FUNCTION_BLOCK "G152M_Code"
TITLE =G152M EXHAUST AIR LOUVER GERM 3
//COPYRIGHT:    (C) 2009  BUHLER AG, CH-9240 UZWIL, SWITZERLAND
//
//PRODUCT:      WinCoS_BIW01_09
//
//TITLE:        EXHAUST AIR LOUVER GERM 3
//                Machine group control
//                Maschinengruppensteuerung
//
//--------------------------------------------------------------------------------
//
//IDENT:        AUTHOR:             DEPT:                              DATE:
//
//P01_FB252.1.0 K.Renz              CSB41                              13.Jan.2010
//             1st Release
//
//--------------------------------------------------------------------------------
//
//PURPOSE:
//
//MANUAL :
//
//RESTRICTIONS:
//
//--------------------------------------------------------------------------------
AUTHOR : KR
FAMILY : USW
VERSION : 9.9


VAR
  Gr : "GCS7_GrpCtrlSub";	//Standard interface to group
  InOutValue1 : DINT ;	//Data for user
  InOutValue2 : DINT ;	//Data for user
  OutWayConflict : BOOL ;	//Data for user
  OutSelectionOk : BOOL ;	//Data for user
  CmdNewValue : BOOL ;	//Data for user
  CmdNewJob : BOOL ;	//Data for user
  OutCodeOK : BOOL ;	//Data for user
  InEndOfJob : BOOL ;	//Data for user
  staWayOk : BOOL ;	//Data for user
  EdgeStartRelease : BOOL ;	//Data for user
  USW8 : BOOL ;	//Data for user
  USW9 : BOOL ;	//Data for user
  USW10 : BOOL ;	//Data for user
  USW11 : BOOL ;	//Data for user
  USW12 : BOOL ;	//Data for user
  USW13 : BOOL ;	//Data for user
  USW14 : BOOL ;	//Data for user
  USW15 : BOOL ;	//Data for user
  A_2350_BZS01 : "GCS7_E_DigInput";	// DigInpCont
  A_2350_BZS02 : "GCS7_E_DigInput";	// DigInpCont
  A_2350_MXZ01 : "GCS7_E_ValveControl4Pos";	// VLS4Ctrl
END_VAR
VAR_TEMP
  tmpEnable : BOOL ;
  tmpFlag : BOOL ;
  tmpCmdNext : BOOL ;
  tmpLocal : BOOL ;
  tmpAspOk : BOOL ;
  tmpHWStop : BOOL ;
  tmpInstanzDBNo : INT ;
END_VAR
BEGIN
NETWORK
TITLE =



NETWORK
TITLE =Read command from group control
//Parameter
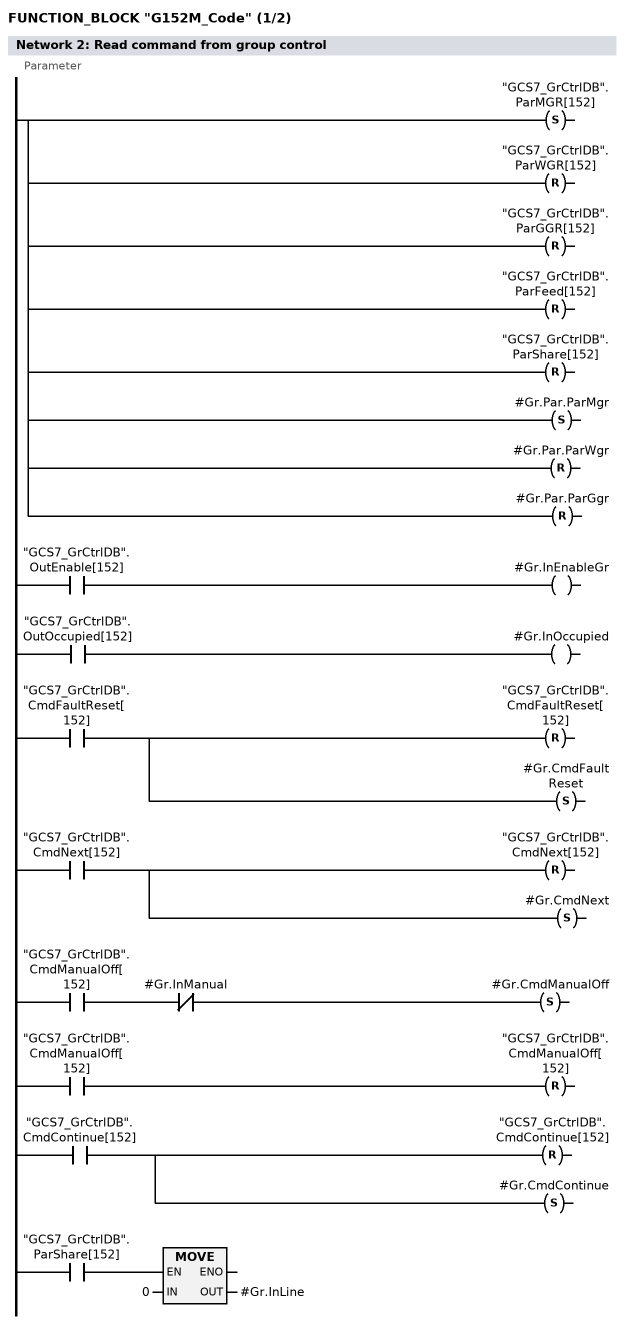
      SET   ;
      S     "GCS7_GrCtrlDB".ParMGR[152];
      R     "GCS7_GrCtrlDB".ParWGR[152];
      R     "GCS7_GrCtrlDB".ParGGR[152];
      R     "GCS7_GrCtrlDB".ParFeed[152];
      R     "GCS7_GrCtrlDB".ParShare[152];
      S     #Gr.Par.ParMgr;
      R     #Gr.Par.ParWgr;
      R     #Gr.Par.ParGgr;
//Command
      U     "GCS7_GrCtrlDB".OutEnable[152];
      =     #Gr.InEnableGr;
      U     "GCS7_GrCtrlDB".OutOccupied[152];
      =     #Gr.InOccupied;
      U     "GCS7_GrCtrlDB".CmdFaultReset[152];
      R     "GCS7_GrCtrlDB".CmdFaultReset[152];
      S     #Gr.CmdFaultReset;
      U     "GCS7_GrCtrlDB".CmdNext[152];
      R     "GCS7_GrCtrlDB".CmdNext[152];
      S     #Gr.CmdNext;

      U     "GCS7_GrCtrlDB".CmdManualOff[152];
      UN    #Gr.InManual;
      S     #Gr.CmdManualOff;
      U     "GCS7_GrCtrlDB".CmdManualOff[152];
      R     "GCS7_GrCtrlDB".CmdManualOff[152];

//      U     "GCS7_GrCtrlDB".CmdManualOff[152]
//      O     "GCS7_GrCtrlDB".OutOccupied[152]
//      R     "GCS7_GrCtrlDB".CmdManualOff[152]
//      S     #Gr.CmdManualOff

      U     "GCS7_GrCtrlDB".CmdContinue[152];
      R     "GCS7_GrCtrlDB".CmdContinue[152];
      S     #Gr.CmdContinue;
//Init Line Number
      U     "GCS7_GrCtrlDB".ParShare[152];
      SPBN  WE00;
      L     0;
      T     #Gr.InLine;
WE00: NOP   0;
NETWORK
TITLE =Call Methode Control
// 1. Handle Interface PCControl
// 2. Prepare mode --> ModePassive,ModeActive,ModeIdling
// 3. Reset global flags of the group
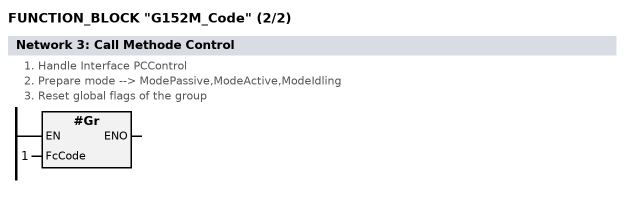
      CALL #Gr (
           FcCode                   := 1);
NETWORK
TITLE =Restart Idling Time

      L     #Gr.Par.ParIdling;
      L     2;
      >=I   ;
      SPB   IdTm;
      T     #Gr.Par.ParIdling;
IdTm: NOP   0;
      CLR   ;
      S     #Gr.CmdRestartIdling;
NETWORK
TITLE =Prepare global flags



NETWORK
TITLE =Set Pattern (Target position)

      U     #Gr.InManual;
      SPB   ILO6;
      L     0; // 0.0%
      O     "MAL1S019".PCRead.Step.StIdling;
      O     "MAL1S019".PCRead.Step.StPassive;
      SPB   PE;
      U     "MAL1S019Par".Par.FlagProcess.ProcessActive;
      O(    ;
      U     "MAL1S019Par".Par.FlagProcess.ProcessEnd; // germinating Process finished
      UN    "MAL1S019".PCRead.Step.StEmptying;
      )     ;
      SPBN  M003;
      NOP   0;
//BRT100310 - Abluftklappen haben gleichen Sollwert wie Frischluftklappen!
//      L     100                         // 100%
//      L     "MAL1S019Par".StepAct.PosWasteAirFlapBasic
//      -I
      L     "MAL1S019Par".Par.ParIntMachine.TargetPosFreshAir; //BRT100310
      L     "MAL1S019Par".Par.ParIntProcess.Value29; // Target Position FreshAir 2
      +I    ;
      L     2;
      /I    ;
      L     10; // convert to 0.1%
      *I    ;
PE:   NOP   0;

      U     "G152M".A_2350_MXZ01.InManual;
      SPB   Man1;
      T     #A_2350_MXZ01.InPositionMiddle; // setpoint element
Man1: NOP   0;

M003: NOP   0;
      SPA   En06;
ILO6: NOP   0;
//BRT100310      L     100                         // 100%
      L     "MAL1S019Par".Par.ParIntProcess.TarPos_ILO_FreshAir;
//BRT100310      -I
      L     10; // convert to 0.1%
      *I    ;
      T     #A_2350_MXZ01.InPositionMiddle; // setpoint element
En06: NOP   0;



NETWORK
TITLE =Interlocking WayOk



NETWORK
TITLE =Interlocking Autostart

      CLR   ;
      R     #Gr.OutAutostart;
NETWORK
TITLE =Interlocking Enable
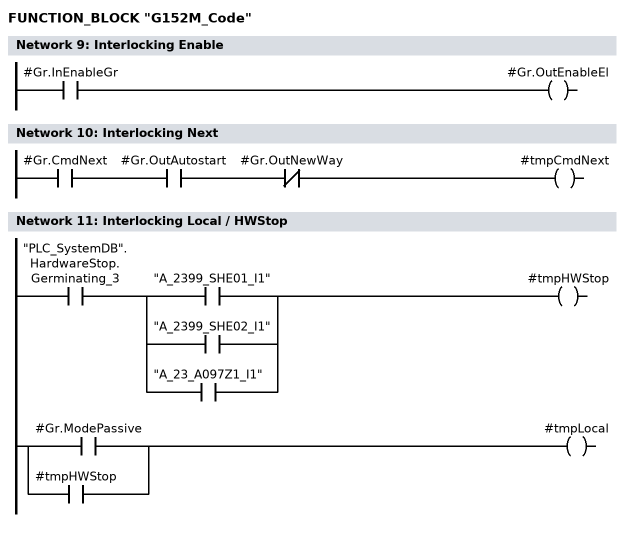

      U     #Gr.InEnableGr;
      =     #Gr.OutEnableEl;

NETWORK
TITLE =Interlocking Next

      U     #Gr.CmdNext;
      U     #Gr.OutAutostart;
      UN    #Gr.OutNewWay;
      =     #tmpCmdNext;

NETWORK
TITLE =Interlocking Local / HWStop

      U     "PLC_SystemDB".HardwareStop.Germinating_3;
//BRT100310 - HW-Stop nur bei NOT-AUS +C23 oder Customer, nicht bei NOT-AUS Maschine!
      U(    ;
      O     "A_2399_SHE01_I1";
      O     "A_2399_SHE02_I1";
      O     "A_23_A097Z1_I1";
      )     ;
      =     #tmpHWStop;

      U     #Gr.ModePassive;
      O     #tmpHWStop;
      =     #tmpLocal;

NETWORK
TITLE ==A-2350-BZS02 : LOUVER EXHAUST AIR 100%  OPEN

      NOP   0;
//-InLocal---
      U     #tmpLocal;
      =     #A_2350_BZS02.InLocal;
//
//-Monitoring---
      CLR   ;
      =     #A_2350_BZS02.InMonTrue;
      CLR   ;
      =     #A_2350_BZS02.InMonFalse;
//
//-PreAlarm---
      CLR   ;
      =     #A_2350_BZS02.InPreAlarmTrue;
      CLR   ;
      =     #A_2350_BZS02.InPreAlarmFalse;
//
//-Additional commands---
//      CLR
//      S     #A_2350_BZS02.CmdRunTimeOutTime
//
//-Read inputs---
      U     "A_2350_BZS02_I1";
      =     #A_2350_BZS02.InpTrue;
      U     "PLC_DPInfo".Master[1].SlavesError[38];
      =     #A_2350_BZS02.InDPFault;
//
//-Set Parameters---
//
//-Call object control---
      CALL #A_2350_BZS02 ;
//
//-Write outputs---
NETWORK
TITLE ==A-2350-BZS01 : LOUVER EXHAUST AIR 0% CLOSED

      NOP   0;
//-InLocal---
      U     #tmpLocal;
      =     #A_2350_BZS01.InLocal;
//
//-Monitoring---
      CLR   ;
      =     #A_2350_BZS01.InMonTrue;
      CLR   ;
      =     #A_2350_BZS01.InMonFalse;
//
//-PreAlarm---
      CLR   ;
      =     #A_2350_BZS01.InPreAlarmTrue;
      CLR   ;
      =     #A_2350_BZS01.InPreAlarmFalse;
//
//-Additional commands---
//      CLR
//      S     #A_2350_BZS01.CmdRunTimeOutTime
//
//-Read inputs---
      U     "A_2350_BZS01_I1";
      =     #A_2350_BZS01.InpTrue;
      U     "PLC_DPInfo".Master[1].SlavesError[38];
      =     #A_2350_BZS01.InDPFault;
//
//-Set Parameters---
//
//-Call object control---
      CALL #A_2350_BZS01 ;
//
//-Write outputs---
NETWORK
TITLE ==A-2350-MXZ01 : LOUVER EXHAUST AIR

      NOP   0;
//-InLocal---
      U(    ;
      U     #tmpLocal;
      O     ;
      U     #Gr.InManual;
      UN    #Gr.InOutAutostartMan;
      )     ;
      U     #A_2350_MXZ01.StLN;
      =     #A_2350_MXZ01.InLocal;

//-Interlocking---
      U     #A_2350_MXZ01.Par.ParManual;
      U     #A_2350_MXZ01.InManual;
      SPB   man1;
      U(    ;
      L     0;
      L     #A_2350_MXZ01.InPositionMiddle; // setpoint element
      ==I   ;
      )     ;
      U(    ;
      U     #Gr.InManual;
      U     #Gr.InOutAutostartMan;
      ON    #Gr.InManual;
      )     ;
      U     #Gr.OutEnableEl;
      =     #A_2350_MXZ01.InLN;

      U(    ;
      L     #A_2350_MXZ01.InPositionMiddle; // setpoint element
      L     0;
      >I    ;
      )     ;
      U(    ;
      L     #A_2350_MXZ01.InPositionMiddle; // setpoint element
      L     1000; // 100,0%
      <I    ;
      )     ;
      U(    ;
      U     #Gr.InManual;
      U     #Gr.InOutAutostartMan;
      ON    #Gr.InManual;
      )     ;
      U     #Gr.OutEnableEl;
      S     #A_2350_MXZ01.CmdMiddle1;

      CLR   ;
      =     #A_2350_MXZ01.CmdMiddle2;

      U(    ;
      UN    #Gr.InOccupied;
      UN    #Gr.InManual;
      )     ;
      O(    ;
      L     #A_2350_MXZ01.InPositionMiddle; // setpoint element
      L     1000; // 100,0%
      >=I   ;
      )     ;
      U(    ;
      U     #Gr.InManual;
      U     #Gr.InOutAutostartMan;
      ON    #Gr.InManual;
      )     ;
      U     #Gr.OutEnableEl;
      S     #A_2350_MXZ01.CmdHN;
man1: NOP   0;
//
//-Read inputs---
//====>BRT100310 - Regeln auf Zeit, ohne Auswertung Rückmeldung
      U     "A_2350_BZS01_I1";
      =     "G152M".A_2350_MXZ01.InpLN;
      CLR   ;
      =     "G152M".A_2350_MXZ01.InpMiddle1;
      U     "A_2350_BZS02_I1";
      =     "G152M".A_2350_MXZ01.InpHN;

//      U     #A_2350_BZS02.StTrue        // 100% Abluft - Klappe OFFEN
//      SPBN  FL1
//      L     1950
//      SPA   INP1
//FL1:  NOP   0
//      U     #A_2350_BZS01.StTrue        // 0% Abluft - Klappe ZU
//      SPBN  RL1
//      L     0
//      SPA   INP1
//RL1:  NOP   0
//      L     "A_2350_BEE01_AI1"
//      L     10
//      /I
//INP1: T     #A_2350_MXZ01.InpPosition
//<====BRT100310
//BRT110310      U     "PLC_SystemDB".HardwareStop.Germinating_3
      U     #tmpHWStop; //BRT110310
      =     #A_2350_MXZ01.InHWStop;
      U     "PLC_DPInfo".Master[1].SlavesError[33];
      O     "PLC_DPInfo".Master[1].SlavesError[38];
      =     #A_2350_MXZ01.InDPFault;
//
//-Set Parameters---
//
//-Call object control---
      CALL #A_2350_MXZ01 ;
//
//-Write outputs---
      U     #A_2350_MXZ01.OutpLN;
      =     "A_2350_MXZ01_O2";
      U     #A_2350_MXZ01.OutpHN;
      =     "A_2350_MXZ01_O1";

NETWORK
TITLE =Test Fault

      U     #A_2350_BZS01.StFault;
      O     #A_2350_BZS02.StFault;
      O     #A_2350_MXZ01.StFault;
      =     #Gr.VarFault;
NETWORK
TITLE =Test Warning

      CLR   ;
      =     #Gr.OutWarning;
NETWORK
TITLE =Test Stopped
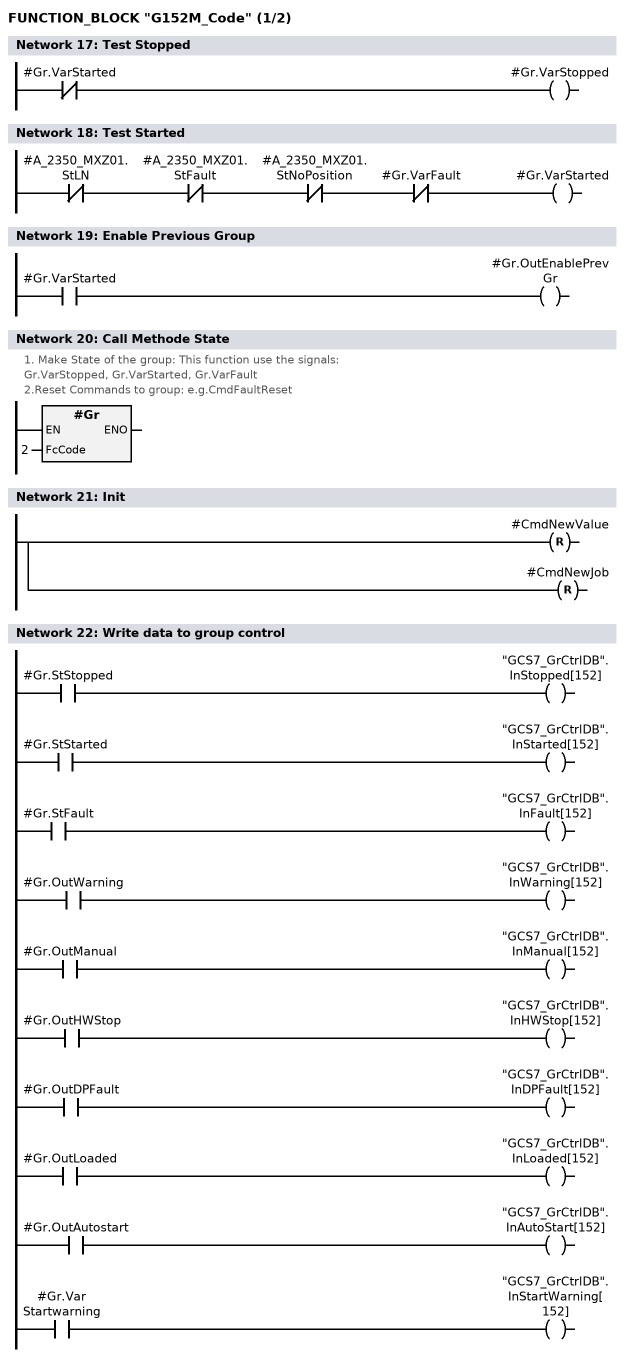

//BRT100310      U     #A_2350_MXZ01.StLN
//BRT100310      UN    #Gr.VarFault
      UN    #Gr.VarStarted;
      =     #Gr.VarStopped;
NETWORK
TITLE =Test Started

      UN    #A_2350_MXZ01.StLN;
      UN    #A_2350_MXZ01.StFault;
      UN    #A_2350_MXZ01.StNoPosition;
//BRT100310      UN    #Gr.VarStopped
      UN    #Gr.VarFault;
      =     #Gr.VarStarted;
NETWORK
TITLE =Enable Previous Group

      U     #Gr.VarStarted;
      =     #Gr.OutEnablePrevGr;
NETWORK
TITLE =Call Methode State
//1. Make State of the group: This function use the signals:
//        Gr.VarStopped, Gr.VarStarted, Gr.VarFault
//2.Reset Commands to group: e.g.CmdFaultReset
      CALL #Gr (
           FcCode                   := 2);
NETWORK
TITLE =Init

      SET   ;
      R     #CmdNewValue;
      R     #CmdNewJob;
NETWORK
TITLE =Write data to group control

      U     #Gr.StStopped;
      =     "GCS7_GrCtrlDB".InStopped[152];
      U     #Gr.StStarted;
      =     "GCS7_GrCtrlDB".InStarted[152];
      U     #Gr.StFault;
      =     "GCS7_GrCtrlDB".InFault[152];
      U     #Gr.OutWarning;
      =     "GCS7_GrCtrlDB".InWarning[152];
      U     #Gr.OutManual;
      =     "GCS7_GrCtrlDB".InManual[152];
      U     #Gr.OutHWStop;
      =     "GCS7_GrCtrlDB".InHWStop[152];
      U     #Gr.OutDPFault;
      =     "GCS7_GrCtrlDB".InDPFault[152];
      U     #Gr.OutLoaded;
      =     "GCS7_GrCtrlDB".InLoaded[152];
      U     #Gr.OutAutostart;
      =     "GCS7_GrCtrlDB".InAutoStart[152];
      U     #Gr.VarStartwarning;
      =     "GCS7_GrCtrlDB".InStartWarning[152];
NETWORK
TITLE =End of block
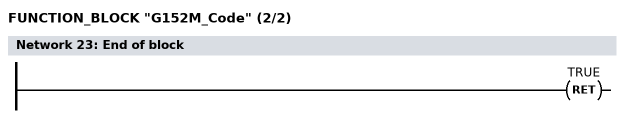

      BE    ;

END_FUNCTION_BLOCK

